PROGRAM Accuracy_Measurement
VAR
	
{region 'Axis Control FB'}	
	fbAxis 						: AXIS_REF;			// Axis to be moved
	
	fbPower						: MC_Power;			// Power the axis
	bPower						: BOOL;
	                			
	fbMove						: MC_MoveAbsolute;  // Move the axis
	bMove						: BOOL;
	fTarget						: LREAL;
	fVelocity					: LREAL := 100;
	fAcceleration				: LREAL;
	fJerk 						: LREAL;
	stOutputs					: ST_McOutputs;
		 
	fPositionError				: LREAL;			// Load Following error
	aRollingBuffer				: ARRAY[1..GVL_AccuracyTest.N_NBR_DELAY_CYCLES] OF LREAL; // Dead time of set pos
		 
	
	fbCompensation				: PositionCompensation_1D;  // Compensation
{endregion}	      	
	 
{region 'Load Position'}
	nLoadPositionRaw AT%I*		: DINT;				// Raw 
	fLoadPositionScaled 		: LREAL;			// Scaled Position in NC unit
	fLoadPositionOffset 		: LREAL := -74.157595; // To be calibrated for the current axis
{endregion}	

{region 'Cycle control'}	
	aSetposition				: ARRAY[1..GVL_AccuracyTest.N_NBR_POSITIONS] OF LREAL; // all positions for the measurement
	aMeasuredData				: ARRAY[1..GVL_AccuracyTest.N_NBR_POSITIONS, 1..2*GVL_AccuracyTest.ciNumCycles] OF LREAL; // Cycles : odd = forward, even = backward
	nCurrentSetpoint 			: UINT;			//
	nCurrentCycle	  			: UINT;
	bBackward					: BOOL;		     // Moving Backward
	fPositionMin				: LREAL := -170; // initialized from the NC
	fPositionMax				: LREAL := 30;   // initialized from the NC
	fStep						: LREAL;
{endregion}

{region 'ISO 230-2 metrics'}	
	aAverageForward					: ARRAY[1..GVL_AccuracyTest.N_NBR_POSITIONS] OF LREAL; 
	aAverageBackward				: ARRAY[1..GVL_AccuracyTest.N_NBR_POSITIONS] OF LREAL; 
	aAverageBidir					: ARRAY[1..GVL_AccuracyTest.N_NBR_POSITIONS] OF LREAL; 
	aSigmaForward					: ARRAY[1..GVL_AccuracyTest.N_NBR_POSITIONS] OF LREAL; 
	aSigmaBackward					: ARRAY[1..GVL_AccuracyTest.N_NBR_POSITIONS] OF LREAL; 
	aReversal						: ARRAY[1..GVL_AccuracyTest.N_NBR_POSITIONS] OF LREAL; 
	fReversalValue					: LREAL;
	aRepeatabilityForward 			: ARRAY[1..GVL_AccuracyTest.N_NBR_POSITIONS] OF LREAL;
	aRepeatabilityBackward 			: ARRAY[1..GVL_AccuracyTest.N_NBR_POSITIONS] OF LREAL;
	aRepeatabilityBidir				: ARRAY[1..GVL_AccuracyTest.N_NBR_POSITIONS] OF LREAL;
	fRepeatForward					: LREAL;
	fRepeatBackWard					: LREAL;
	fRepeatBidir					: LREAL;
	fSystematicAccuracyForward 		: LREAL;
	fSystematicAccuracyBackward		: LREAL;
	fSystematicAccuracyBidir 		: LREAL;
	fAverageBidirError				: LREAL;
	fAccuracyForward 				: LREAL;
	fAccuracyBackward 				: LREAL;
	fAccuracyBidir					: LREAL;	
{endregion}
	

          			

{region 'Inialization'}                			
	fScalingNum					: LREAL;
	fScalingDenum				: LREAL;
	                    		
	fbReadAccel					: MC_ReadParameter;
	fbReadJerk					: MC_ReadParameter;
	fbReadScalingNum			: MC_ReadParameter;
	fbReadScalingDenum			: MC_ReadParameter;
	fbReadMinPos				: MC_ReadParameter;
	fbReadMaxPos				: MC_ReadParameter;	 
{endregion}
	 
	
{region 'commands of the program'} 
	
	{attribute 'init_on_onlchange' }
	bInit						: BOOL;					// Start the initalization
	{attribute 'init_on_onlchange' }
	bRead						: BOOL;					// Read the init data			
	
	bStartMeasure				: BOOL;					// Start the accuracy measurement cycle
	nStateMeasure				: E_Aquisition_State;
	
	bCompute					: BOOL;					// Start the metrics computation
	
	bTestAccuracy 				: BOOL;					// Execute the cycle without measurement
	nStateTestAccuracy			: E_TestAccuracy_State;
		 
	bStop 						: BOOL;					// Stop cycles
	
	// Data for Scope Display
	fDisplaySetpointForward, fDisplaySetpointBackward, fDisplayMeasurementForward, fDisplayMeasurementBackward 	: LREAL;
	fDisplaySetpointComput, fDisplayMeasurementAverageForward, fDisplayMeasurementAverageBackward 				: LREAL;
	
	bCompensate					: BOOL;					// Start usung the compensation
{endregion}	

	

END_VAR

// Don't go further if not init
IF NOT bInit THEN
	 bRead := TRUE;
	 Init();
	 RETURN;
END_IF


//Start Acquistion
IF bStartMeasure THEN
	IF fbAxis.Status.Disabled THEN
		bPower := TRUE;
	ELSE
		nCurrentCycle := 0;
		nCurrentSetpoint := 1;
		nStateMeasure := E_Aquisition_State.MOVE_TO_FIRST_POS;
		bStartMeasure := FALSE;
	END_IF
END_IF

//Start Measurement
IF bTestAccuracy THEN
	IF fbAxis.Status.Disabled THEN
		bPower := TRUE;
	ELSE
		nCurrentSetpoint := 1;
		nStateTestAccuracy := E_TestAccuracy_State.MOVE_TO_FIRST_POS;
		bTestAccuracy := FALSE;
	END_IF
END_IF

// Compute the metrics
IF bCompute THEN
	bCompute := FALSE;
	Compute();
END_IF


// Cyclic Update
Cycle();
Acquisition();
TestAccuracy();

METHOD Acquisition : BOOL
(* This method moves the axis and aquires the position data to be processed later in the compute method *)

CASE nStateMeasure OF
	E_Aquisition_State.IDLE: // IDLE
		;
		
	E_Aquisition_State.MOVE_TO_FIRST_POS:
		fTarget := fPositionMin;
		bMove := TRUE;
		nStateMeasure := E_Aquisition_State.WAIT_MOVE_TO_FIRST_POS;
		
	E_Aquisition_State.WAIT_MOVE_TO_FIRST_POS:
		IF stOutputs.Done THEN
			bMove := FALSE;
			nStateMeasure :=  E_Aquisition_State.MOVE_TO_TARGET_FORWARD;
			nCurrentCycle	 := nCurrentCycle+1;
			nCurrentSetpoint := 1;
		END_IF
		
		IF nCurrentCycle > 2*GVL_AccuracyTest.N_NBR_CYCLES THEN
			nStateMeasure :=  E_Aquisition_State.DONE;
		END_IF
		
	E_Aquisition_State.MOVE_TO_TARGET_FORWARD:
		fTarget := aSetposition[nCurrentSetpoint];
		bMove := TRUE;
		nStateMeasure := E_Aquisition_State.WAIT_MOVE_TO_TARGET_FORWARD;
		
	E_Aquisition_State.WAIT_MOVE_TO_TARGET_FORWARD:
		IF stOutputs.Done  THEN
			bMove := FALSE;
			aMeasuredData[nCurrentSetpoint,nCurrentCycle] := fLoadPositionScaled-aSetposition[nCurrentSetpoint];
			fDisplayMeasurementForward := aMeasuredData[nCurrentSetpoint,nCurrentCycle];
			fDisplaySetpointForward := aSetposition[nCurrentSetpoint];
			nStateMeasure := E_Aquisition_State.MOVE_TO_TARGET_FORWARD;
			nCurrentSetpoint := nCurrentSetpoint+1;		
		END_IF
		IF nCurrentSetpoint > GVL_AccuracyTest.N_NBR_POSITIONS THEN
			nStateMeasure := E_Aquisition_State.MOVE_TO_LAST_POS;
		END_IF
		
	E_Aquisition_State.MOVE_TO_LAST_POS : 
		fTarget := fPositionMax;
		bMove := TRUE;
		nStateMeasure := E_Aquisition_State.WAIT_MOVE_TO_LAST_POS;	
	
	E_Aquisition_State.WAIT_MOVE_TO_LAST_POS:
		IF stOutputs.Done THEN
			bMove := FALSE;
			nStateMeasure := E_Aquisition_State.WAIT_MOVE_TO_TARGET_BACKWARD;
			nCurrentSetpoint := GVL_AccuracyTest.N_NBR_POSITIONS;
			nCurrentCycle	 := nCurrentCycle+1;
		END_IF		
		IF nCurrentCycle > 2*GVL_AccuracyTest.N_NBR_CYCLES THEN
			nStateMeasure := E_Aquisition_State.DONE;
		END_IF
		
	E_Aquisition_State.MOVE_TO_TARGET_BACKWARD:
		fTarget := aSetposition[nCurrentSetpoint];
		bMove := TRUE;
		nStateMeasure := E_Aquisition_State.WAIT_MOVE_TO_TARGET_BACKWARD;
		
	E_Aquisition_State.WAIT_MOVE_TO_TARGET_BACKWARD:
		IF stOutputs.Done  THEN
			bMove := FALSE;
			aMeasuredData[nCurrentSetpoint,nCurrentCycle] := fLoadPositionScaled-aSetposition[nCurrentSetpoint];
			fDisplayMeasurementBackward := aMeasuredData[nCurrentSetpoint,nCurrentCycle];
			fDisplaySetpointBackward := aSetposition[nCurrentSetpoint];
			nStateMeasure := E_Aquisition_State.MOVE_TO_TARGET_BACKWARD;
			nCurrentSetpoint := nCurrentSetpoint-1;		
		END_IF
		IF nCurrentSetpoint < 1 THEN
			nStateMeasure := E_Aquisition_State.MOVE_TO_FIRST_POS;
		END_IF
		
	E_Aquisition_State.DONE:
		bCompute := TRUE;
		nStateMeasure := E_Aquisition_State.IDLE;

END_CASE
END_METHOD

METHOD Compute : BOOL
VAR
	i , j : UINT;
	aTempDataForward : ARRAY[1..GVL_AccuracyTest.N_NBR_CYCLES] OF LREAL;
	aTempDataBackward : ARRAY[1..GVL_AccuracyTest.N_NBR_CYCLES] OF LREAL;
	lrMaxForward		: LREAL;
	lrMinForward		: LREAL;
	lrMaxBackward		: LREAL;
	lrMinBackward		: LREAL;
END_VAR
(* This method computes the positioning accuracy metrics according to ISO 230-2 *)

// ***** initialization ******** //
lrMinForward  := 1E300;
lrMinBackward := 1E300;
lrMaxForward := -1E300;
lrMaxBackward := -1E300;

// ***** compute data for all positions  ******** //
FOR i := 1 TO GVL_AccuracyTest.N_NBR_POSITIONS DO
	// gather all samples for each position
	FOR j := 1 TO GVL_AccuracyTest.N_NBR_CYCLES DO
		aTempDataForward[j] := aMeasuredData[i,2*j-1];
		aTempDataBackward[j] := aMeasuredData[i,2*j];
	END_FOR
	
	// compute the average at this position
	aAverageForward[i] := average(aTempDataForward);
	aAverageBackward[i] := average(aTempDataBackward);
	aAverageBidir[i] := (aAverageForward[i]+aAverageBackward[i])/2;
	
	// compute the reversal value  at this position
	aReversal[i] := aAverageForward[i]-aAverageBackward[i];
	
	// compute the standard deviation at this position
	aSigmaForward[i] := sigma(aTempDataForward,aAverageForward[i]);
	aSigmaBackward[i] := sigma(aTempDataBackward,aAverageBackward[i]);
	
	// find the extremities of each travel
	lrMaxForward	:= MAX(lrMaxForward,aAverageForward[i]+2*aSigmaForward[i] );
	lrMinForward	:= MIN(lrMinForward,aAverageForward[i]-2*aSigmaForward[i] );
	lrMaxBackward	:= MAX(lrMaxBackward,aAverageBackward[i]+2*aSigmaBackward[i] );
	lrMinBackward   := MIN(lrMinBackward,aAverageBackward[i]-2*aSigmaBackward[i] );
	
	// compute the repeatability for each value
	aRepeatabilityForward[i] := 4*aSigmaForward[i];
	aRepeatabilityBackward[i] := 4*aSigmaBackward[i];
	aRepeatabilityBidir[i] := MAX(2*aSigmaForward[i]+2*aSigmaBackward[i]+ABS(aReversal[i]),aRepeatabilityForward[i],aRepeatabilityBackward[i]);
END_FOR


// ***** compute the metrics ******** //
//  Reversal value (maximum backlash)
fReversalValue := max_abs_array(aReversal);
// Repeatability
fRepeatForward	 := max_abs_array(aRepeatabilityForward);
fRepeatBackWard := max_abs_array(aRepeatabilityBackward);
fRepeatBidir	 := max_abs_array(aRepeatabilityBidir);
// Systematic accuracy (maximal compensation)
fSystematicAccuracyForward := max_array(aAverageForward) - min_array(aAverageForward) ;
fSystematicAccuracyBackward := max_array(aAverageBackward) - min_array(aAverageBackward) ;
fSystematicAccuracyBidir := MAX(max_array(aAverageForward),max_array(aAverageBackward)) - MIN(min_array(aAverageForward),min_array(aAverageBackward));
// Average Bidirectional error 
fAverageBidirError			:= max_array(aAverageBidir) - min_array(aAverageBidir);
//Reversal value
fAccuracyForward 	:= lrMaxForward-lrMinForward;
fAccuracyBackward 	:= lrMaxBackward- lrMinBackward;
fAccuracyBidir		:= MAX(lrMaxForward,lrMaxBackward)-MIN(lrMinForward,lrMinBackward);

// ***** OPTIONAL start the compensation using this data ******** //
// xCompensate := TRUE;
END_METHOD

METHOD Cycle : BOOL
VAR
	i : DINT;
END_VAR
(* This method takes care of cyclic updates *)

// Keep the axis status up to date
fbAxis.ReadStatus();

// Manage power of the motor
fbPower(
	Axis:= fbAxis, 
	Enable:= bPower, 
	Enable_Positive:= TRUE, 
	Enable_Negative:= TRUE, 
	Override:= 100, 
	BufferMode:= , 
	Options:= , 
	Status=> , 
	Busy=> , 
	Error=> , 
	ErrorID=> );

// Manage the move absolute command
fbMove(
	Axis:= fbAxis, 
	Execute:= bMove, 
	Position:= fTarget, 
	Velocity:= fVelocity, 
	Acceleration:= fAcceleration, 
	Deceleration:= fAcceleration, 
	Jerk:= fJerk, 
	BufferMode:= , 
	Options:= , 
	Done=> stOutputs.Done, 
	Busy=> stOutputs.Busy, 
	Active=> stOutputs.Active, 
	CommandAborted=> stOutputs.CommandAborted, 
	Error=> stOutputs.Error, 
	ErrorID=> stOutputs.ErrorID);
	
// Compensate the accuracy
fbCompensation(
	afCompensationTableForward:= aAverageForward, 
	afCompensationTableBackward:= aAverageBackward, 
	fbAxis:= fbAxis, 
	fStartPosition:= aSetposition[1], 
	fStopPosition:= aSetposition[GVL_AccuracyTest.N_NBR_POSITIONS], 
	bEnable:= bCompensate);
	
//	Load position 
fLoadPositionScaled := Scaling(fInput := nLoadPositionRaw, fScalingNum := fScalingNum, fScalingDenum := fScalingDenum) + fLoadPositionOffset;

// Dead time of the Set Position computed in the PLC 
FOR i := 1 TO  3 DO
	aRollingBuffer[i] := aRollingBuffer[i+1];
END_FOR
aRollingBuffer[i] := fbAxis.NcToPlc.SetPos;

// Load following error
fPositionError := aRollingBuffer[1] - fLoadPositionScaled ;
END_METHOD

METHOD Init : BOOL
VAR
	bValid : BOOL := TRUE;
END_VAR
(* This method reads initialization data from the NC Axis directly *)

bValid := TRUE; 

// Init the acceleration value
fbReadAccel(
	Axis:= fbAxis, 
	Enable:= bRead, 
	ParameterNumber:= MC_AxisParameter.AxisAcc, 
	ReadMode:= E_ReadMode.READMODE_CYCLIC, 
	Valid=> , 
	Busy=> , 
	Error=> , 
	ErrorID=> , 
	Value=> fAcceleration);	
	bValid := bValid AND fbReadAccel.Valid;

// Init the jerk value
fbReadJerk(
	Axis:= fbAxis, 
	Enable:= bRead, 
	ParameterNumber:= MC_AxisParameter.AxisJerk, 
	ReadMode:= E_ReadMode.READMODE_CYCLIC, 
	Valid=> , 
	Busy=> , 
	Error=> , 
	ErrorID=> , 
	Value=> fJerk);	
	bValid := bValid AND fbReadJerk.Valid;
	
// Read the denominator scaling value
fbReadScalingDenum(
	Axis:= fbAxis, 
	Enable:= bRead, 
	ParameterNumber:= MC_AxisParameter.AxisEncoderScalingDenominator, 
	ReadMode:= E_ReadMode.READMODE_CYCLIC, 
	Valid=> , 
	Busy=> , 
	Error=> , 
	ErrorID=> , 
	Value=> fScalingDenum);	
	bValid := bValid AND fbReadScalingDenum.Valid;

// Read the numerator scaling value
fbReadScalingNum(
	Axis:= fbAxis, 
	Enable:= bRead, 
	ParameterNumber:= MC_AxisParameter.AxisEncoderScalingNumerator, 
	ReadMode:= E_ReadMode.READMODE_CYCLIC, 
	Valid=> , 
	Busy=> , 
	Error=> , 
	ErrorID=> , 
	Value=> fScalingNum);	
	bValid := bValid AND fbReadScalingNum.Valid;

// Read the minimum position
fbReadMinPos(
	Axis:= fbAxis, 
	Enable:= bRead, 
	ParameterNumber:= MC_AxisParameter.AxisMinSoftPosLimit , 
	ReadMode:= E_ReadMode.READMODE_CYCLIC, 
	Valid=> , 
	Busy=> , 
	Error=> , 
	ErrorID=> , 
	Value=> fPositionMin);
	bValid := bValid AND fbReadMinPos.Valid;
	
// Read the maximal position
fbReadMaxPos(
	Axis:= fbAxis, 
	Enable:= bRead, 
	ParameterNumber:= MC_AxisParameter.AxisMaxSoftPosLimit, 
	ReadMode:= E_ReadMode.READMODE_CYCLIC, 
	Valid=> , 
	Busy=> , 
	Error=> , 
	ErrorID=> , 
	Value=> fPositionMax);
	bValid := bValid AND fbReadMaxPos.Valid;

	
// If all data is valid, we initialize the steps where the data will be aquired
// NOTE : we should add a random part for the positions, in order to comply with the norm ISO 230-2	but this is not done here
IF bValid THEN
	fStep := (fPositionMax-fPositionMin)/ UINT_TO_LREAL(GVL_AccuracyTest.N_NBR_POSITIONS +1);
	FOR nCurrentSetpoint := 1 TO GVL_AccuracyTest.N_NBR_POSITIONS DO
		aSetposition[nCurrentSetpoint] := fStep*UINT_TO_LREAL(nCurrentSetpoint) + fPositionMin;
	END_FOR
	bInit := TRUE;
	bRead := FALSE;
END_IF
END_METHOD

METHOD TestAccuracy : BOOL
(* This method moves the axis without aquiring the position data *)

CASE nStateTestAccuracy OF
	
	E_TestAccuracy_State.IDLE: // IDLE
		;
		
	E_TestAccuracy_State.MOVE_TO_FIRST_POS:
		fTarget := fPositionMin;
		bMove := TRUE;
		nStateTestAccuracy := E_TestAccuracy_State.WAIT_MOVE_TO_FIRST_POS;
		
	E_TestAccuracy_State.WAIT_MOVE_TO_FIRST_POS:
		IF stOutputs.Done THEN						
			bMove := FALSE;
			nStateTestAccuracy := E_TestAccuracy_State.MOVE_TO_TARGET_FORWARD;
			nCurrentSetpoint := 1;
		END_IF
		
		IF bStop THEN 
			nStateTestAccuracy := E_TestAccuracy_State.DONE;
		END_IF
		
	E_TestAccuracy_State.MOVE_TO_TARGET_FORWARD:
		fTarget := aSetposition[nCurrentSetpoint];
		bMove := TRUE;
		nStateTestAccuracy := E_TestAccuracy_State.WAIT_MOVE_TO_TARGET_FORWARD;
		
	E_TestAccuracy_State.WAIT_MOVE_TO_TARGET_FORWARD:
		IF stOutputs.Done  THEN
			bMove := FALSE;
			nStateTestAccuracy := E_TestAccuracy_State.MOVE_TO_TARGET_FORWARD;
			nCurrentSetpoint := nCurrentSetpoint+1;		
		END_IF
		IF nCurrentSetpoint > GVL_AccuracyTest.N_NBR_POSITIONS THEN
			nStateTestAccuracy := E_TestAccuracy_State.MOVE_TO_LAST_POS;
		END_IF
		
	E_TestAccuracy_State.MOVE_TO_LAST_POS : 
		fTarget := fPositionMax;
		bMove := TRUE;
		nStateTestAccuracy := E_TestAccuracy_State.WAIT_MOVE_TO_LAST_POS;	
	
	E_TestAccuracy_State.WAIT_MOVE_TO_LAST_POS:
		IF stOutputs.Done THEN
			bMove := FALSE;
			nStateTestAccuracy := E_TestAccuracy_State.MOVE_TO_TARGET_BACKWARD;
			nCurrentSetpoint := GVL_AccuracyTest.N_NBR_POSITIONS;
		END_IF		
		IF bStop THEN
			nStateTestAccuracy := E_TestAccuracy_State.DONE;
		END_IF
		
	E_TestAccuracy_State.MOVE_TO_TARGET_BACKWARD:
		fTarget := aSetposition[nCurrentSetpoint];
		bMove := TRUE;
		nStateTestAccuracy := E_TestAccuracy_State.WAIT_MOVE_TO_TARGET_BACKWARD;
		
	E_TestAccuracy_State.WAIT_MOVE_TO_TARGET_BACKWARD:
		IF stOutputs.Done  THEN
			bMove := FALSE;
			nStateTestAccuracy := E_TestAccuracy_State.MOVE_TO_TARGET_BACKWARD;
			nCurrentSetpoint := nCurrentSetpoint-1;		
		END_IF
		IF nCurrentSetpoint < 1 THEN
			nStateTestAccuracy := E_TestAccuracy_State.MOVE_TO_FIRST_POS;
		END_IF
		
	E_TestAccuracy_State.DONE:
		nStateTestAccuracy := E_TestAccuracy_State.IDLE;

END_CASE
END_METHOD

END_PROGRAM

(* stored: Version 1.1.0.1, ProductVersion 3.1.4024.12
   POU Accuracy_Measurement: Id {a01ecdcf-7a38-4bbc-8390-526c0b12f84d}, SpecialFunc None
   Method Acquisition: Id {30e62b89-0e2b-4358-b111-ef4f65aa8f1e}
   Method Compute: Id {e10d33ae-779a-4788-b1a2-62df5e2f066d}
   Method Cycle: Id {eec0348b-d7b9-4aab-99ab-629f89df70b9}
   Method Init: Id {6e174f89-7746-43b9-90f0-e09087eedb90}
   Method TestAccuracy: Id {c7c95391-32a9-4e51-b913-fa92db878469} *)
